Universal Robots PolyScope program: gripper instruction.urp

Program gripper instruction (installation=default directory=/programs/hanoi createdIn=5.15.1 lastSavedIn=5.15.1 robotSerialNumber=20245300277)
Calibrated DH parameters: a=[-0.000123, -0.242651, -0.197609, 0.000101, -0.000134, 0]; d=[0.151783, 2.720328, 8.544006, -11.133313, 0.085187, 0.091754]; alpha=[1.570905, -0.007647, 0.007134, 1.569752, -1.572297, 0]; deltaTheta=[0, -0.085522, 6.754906, -0.386214, 0.000017, 0]
InitVariablesNode
Robot Program (runOnlyOnce=false)
  URCap Gripper Activate (Robotiq_Grippers, Robotiq Inc.) dataModel(ResetAndActivateKey=false)
  URCap Gripper (Robotiq_Grippers, Robotiq Inc.) dataModel(position=0.0, force=100.0, speed=100.0, positionInDouble=0.0, forceInDouble=100.0, speedInDouble=100.0, slaveIds=[9], blocking=true)
  URCap Gripper (Robotiq_Grippers, Robotiq Inc.) dataModel(position=100.0, force=100.0, speed=100.0, positionInDouble=100.0, forceInDouble=100.0, speedInDouble=100.0, slaveIds=[9], blocking=true)
  URCap Gripper (Robotiq_Grippers, Robotiq Inc.) dataModel(position=50.0, force=100.0, speed=100.0, positionInDouble=50.0, forceInDouble=100.0, speedInDouble=100.0, slaveIds=[9], blocking=true)
  If 
    Placeholder
  Force Simple feature=Base; selection=[0, 0, 1, 0, 0, 0]; wrench=[0, 0, 0.5, 0, 0, 0]; limitsForce=[0.15, 0.15, 0.15, 1.047198, 1.047198, 1.047198]; limitsMotion=[0.1, 0.1, 0.1, 0.349066, 0.349066, 0.349066]
    Halt
